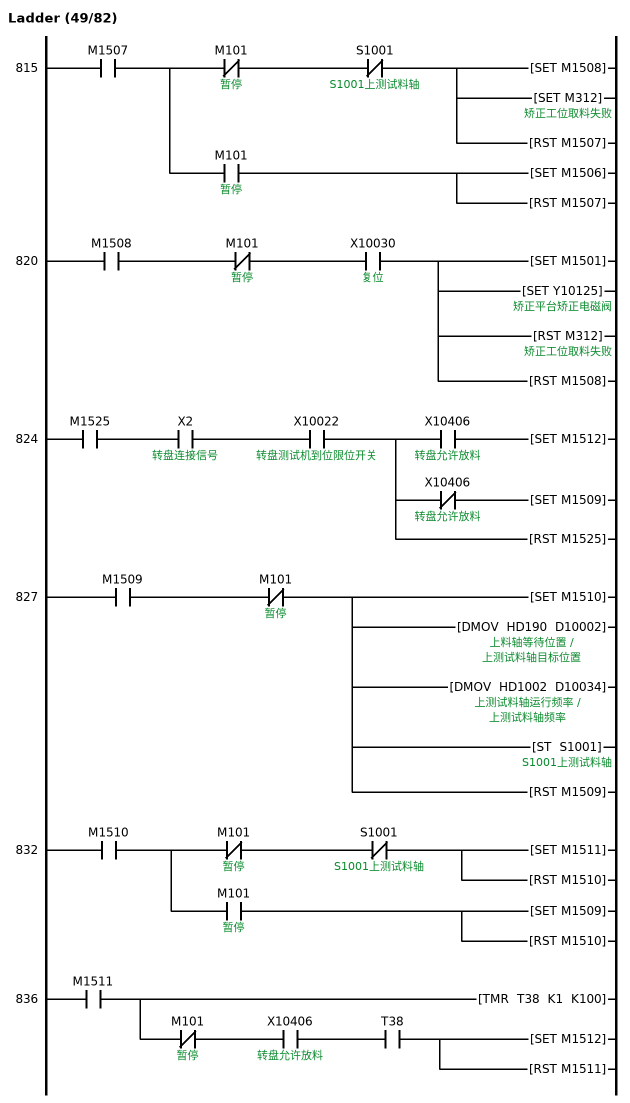
[picture p48: Ladder rows 815-836]
LD     M1507
MPS
ANI    M101	; 暂停
ANI    S1001	; S1001上测试料轴
SET    M1508
SET    M312	; 矫正工位取料失败
RST    M1507
MPP
AND    M101	; 暂停
SET    M1506
RST    M1507
LD     M1508
ANI    M101	; 暂停
AND    X10030	; 复位
SET    M1501
SET    Y10125	; 矫正平台矫正电磁阀
RST    M312	; 矫正工位取料失败
RST    M1508
LD     M1525
AND    X2	; 转盘连接信号
AND    X10022	; 转盘测试机到位限位开关
MPS
AND    X10406	; 转盘允许放料
SET    M1512
MRD
ANI    X10406	; 转盘允许放料
SET    M1509
MPP
RST    M1525
LD     M1509
ANI    M101	; 暂停
SET    M1510
DMOV   HD190 D10002	; 上料轴等待位置 / 上测试料轴目标位置
DMOV   HD1002 D10034	; 上测试料轴运行频率 / 上测试料轴频率
ST     S1001	; S1001上测试料轴
RST    M1509
LD     M1510
MPS
ANI    M101	; 暂停
ANI    S1001	; S1001上测试料轴
SET    M1511
RST    M1510
MPP
AND    M101	; 暂停
SET    M1509
RST    M1510
LD     M1511
TMR    T38 K1 K100
ANI    M101	; 暂停
AND    X10406	; 转盘允许放料
AND    T38
SET    M1512
RST    M1511

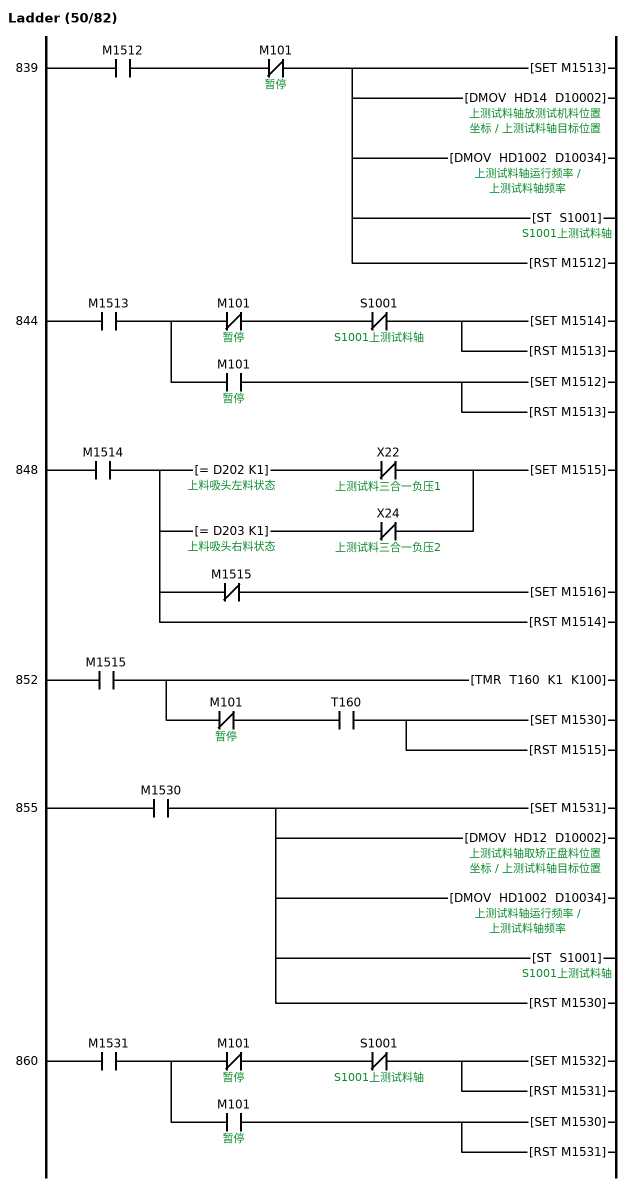
LD     M1512
ANI    M101	; 暂停
SET    M1513
DMOV   HD14 D10002	; 上测试料轴放测试机料位置坐标 / 上测试料轴目标位置
DMOV   HD1002 D10034	; 上测试料轴运行频率 / 上测试料轴频率
ST     S1001	; S1001上测试料轴
RST    M1512
LD     M1513
MPS
ANI    M101	; 暂停
ANI    S1001	; S1001上测试料轴
SET    M1514
RST    M1513
MPP
AND    M101	; 暂停
SET    M1512
RST    M1513
LD     M1514
MPS
LD=    D202 K1	; 上料吸头左料状态
ANI    X22	; 上测试料三合一负压1
LD=    D203 K1	; 上料吸头右料状态
ANI    X24	; 上测试料三合一负压2
ORB
ANB
SET    M1515
MRD
ANI    M1515
SET    M1516
MPP
RST    M1514
LD     M1515
TMR    T160 K1 K100
ANI    M101	; 暂停
AND    T160
SET    M1530
RST    M1515
LD     M1530
SET    M1531
DMOV   HD12 D10002	; 上测试料轴取矫正盘料位置坐标 / 上测试料轴目标位置
DMOV   HD1002 D10034	; 上测试料轴运行频率 / 上测试料轴频率
ST     S1001	; S1001上测试料轴
RST    M1530
LD     M1531
MPS
ANI    M101	; 暂停
ANI    S1001	; S1001上测试料轴
SET    M1532
RST    M1531
MPP
AND    M101	; 暂停
SET    M1530
RST    M1531

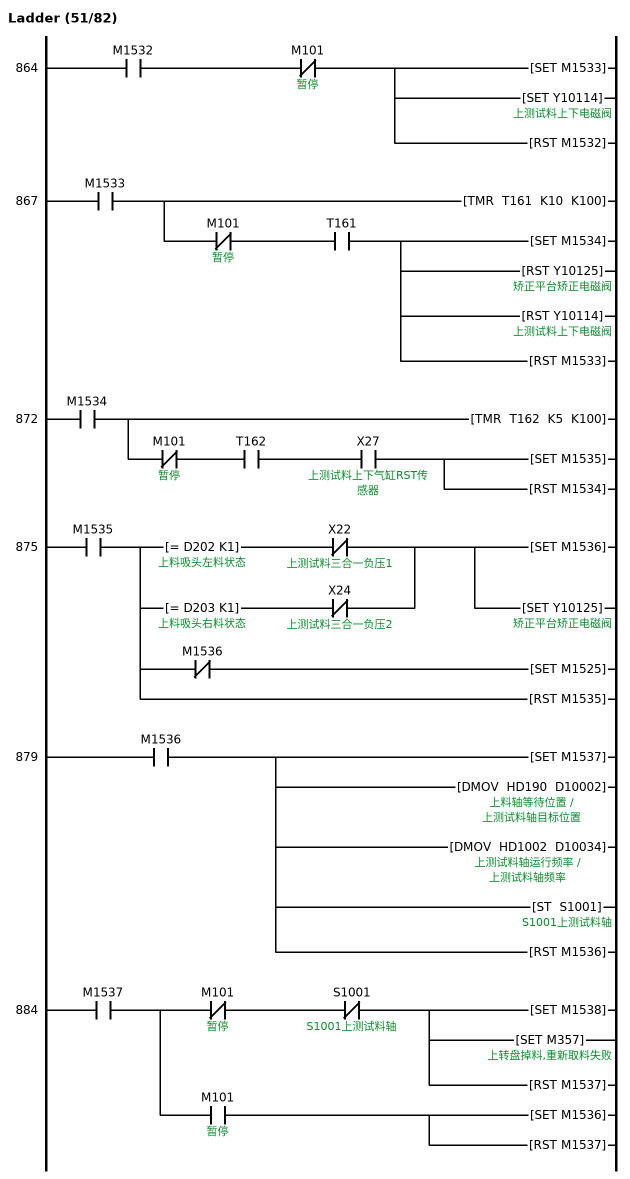
LD     M1532
ANI    M101	; 暂停
SET    M1533
SET    Y10114	; 上测试料上下电磁阀
RST    M1532
LD     M1533
TMR    T161 K10 K100
ANI    M101	; 暂停
AND    T161
SET    M1534
RST    Y10125	; 矫正平台矫正电磁阀
RST    Y10114	; 上测试料上下电磁阀
RST    M1533
LD     M1534
TMR    T162 K5 K100
ANI    M101	; 暂停
AND    T162
AND    X27	; 上测试料上下气缸RST传感器
SET    M1535
RST    M1534
LD     M1535
MPS
LD=    D202 K1	; 上料吸头左料状态
ANI    X22	; 上测试料三合一负压1
LD=    D203 K1	; 上料吸头右料状态
ANI    X24	; 上测试料三合一负压2
ORB
ANB
SET    M1536
SET    Y10125	; 矫正平台矫正电磁阀
MRD
ANI    M1536
SET    M1525
MPP
RST    M1535
LD     M1536
SET    M1537
DMOV   HD190 D10002	; 上料轴等待位置 / 上测试料轴目标位置
DMOV   HD1002 D10034	; 上测试料轴运行频率 / 上测试料轴频率
ST     S1001	; S1001上测试料轴
RST    M1536
LD     M1537
MPS
ANI    M101	; 暂停
ANI    S1001	; S1001上测试料轴
SET    M1538
SET    M357	; 上转盘掉料,重新取料失败
RST    M1537
MPP
AND    M101	; 暂停
SET    M1536
RST    M1537

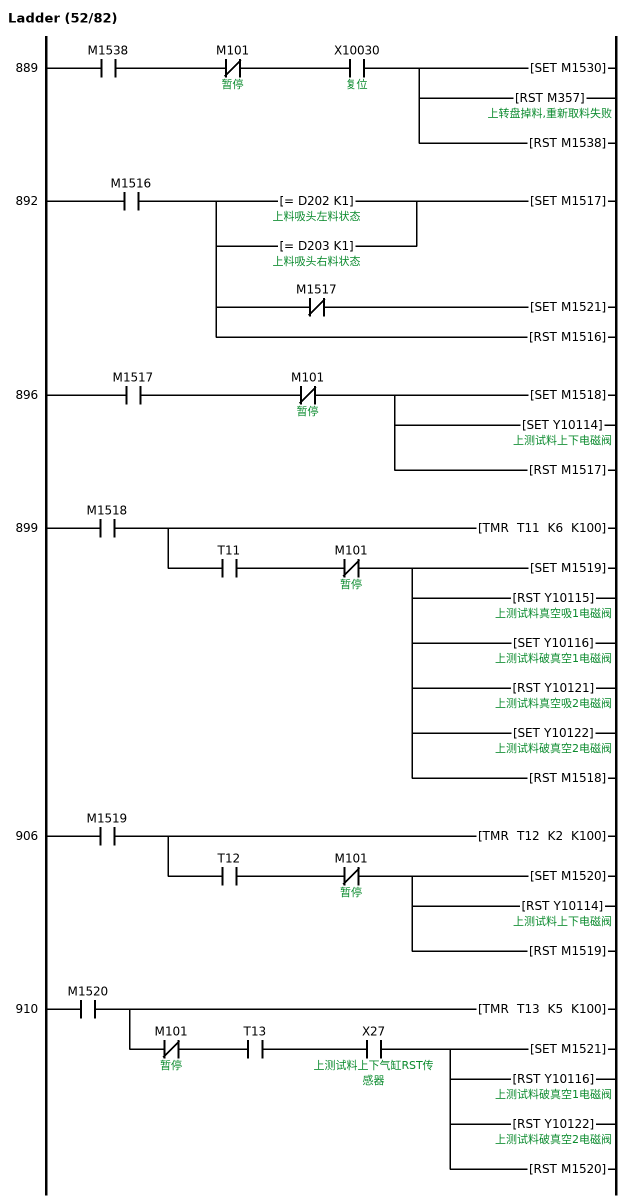
LD     M1538
ANI    M101	; 暂停
AND    X10030	; 复位
SET    M1530
RST    M357	; 上转盘掉料,重新取料失败
RST    M1538
LD     M1516
MPS
LD=    D202 K1	; 上料吸头左料状态
OR=    D203 K1	; 上料吸头右料状态
ANB
SET    M1517
MRD
ANI    M1517
SET    M1521
MPP
RST    M1516
LD     M1517
ANI    M101	; 暂停
SET    M1518
SET    Y10114	; 上测试料上下电磁阀
RST    M1517
LD     M1518
TMR    T11 K6 K100
AND    T11
ANI    M101	; 暂停
SET    M1519
RST    Y10115	; 上测试料真空吸1电磁阀
SET    Y10116	; 上测试料破真空1电磁阀
RST    Y10121	; 上测试料真空吸2电磁阀
SET    Y10122	; 上测试料破真空2电磁阀
RST    M1518
LD     M1519
TMR    T12 K2 K100
AND    T12
ANI    M101	; 暂停
SET    M1520
RST    Y10114	; 上测试料上下电磁阀
RST    M1519
LD     M1520
TMR    T13 K5 K100
ANI    M101	; 暂停
AND    T13
AND    X27	; 上测试料上下气缸RST传感器
SET    M1521
RST    Y10116	; 上测试料破真空1电磁阀
RST    Y10122	; 上测试料破真空2电磁阀
RST    M1520

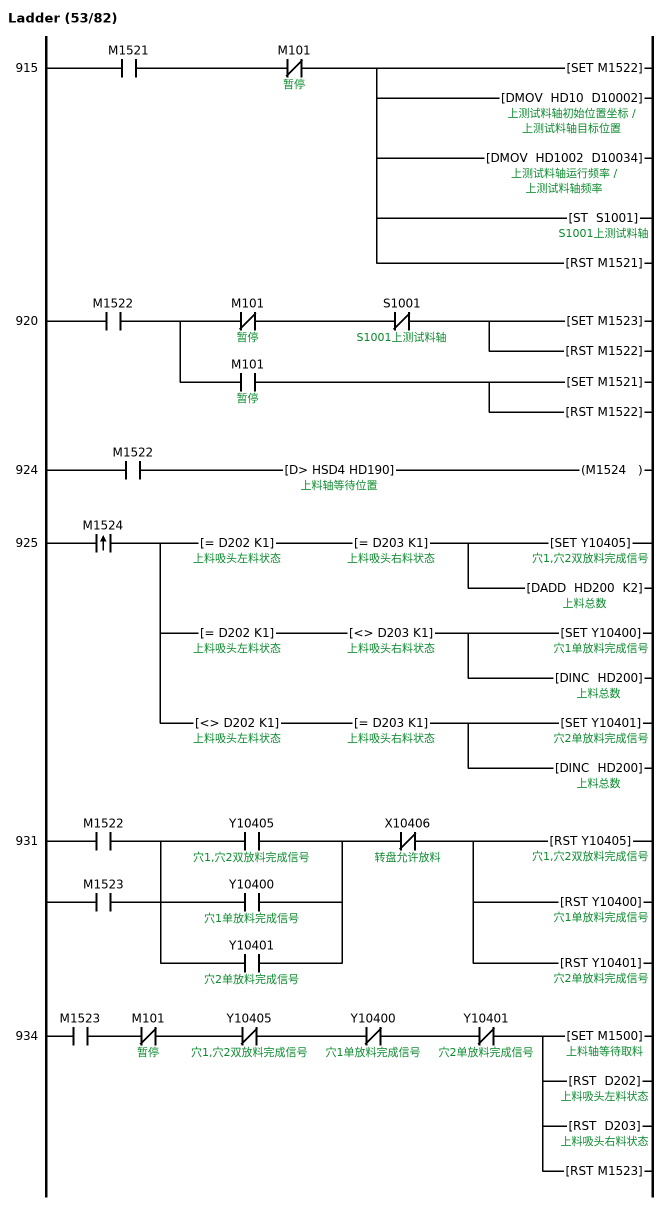
LD     M1521
ANI    M101	; 暂停
SET    M1522
DMOV   HD10 D10002	; 上测试料轴初始位置坐标 / 上测试料轴目标位置
DMOV   HD1002 D10034	; 上测试料轴运行频率 / 上测试料轴频率
ST     S1001	; S1001上测试料轴
RST    M1521
LD     M1522
MPS
ANI    M101	; 暂停
ANI    S1001	; S1001上测试料轴
SET    M1523
RST    M1522
MPP
AND    M101	; 暂停
SET    M1521
RST    M1522
LD     M1522
DAND>  HSD4 HD190	; 上料轴等待位置
OUT    M1524
LDP    M1524
MPS
AND=   D202 K1	; 上料吸头左料状态
AND=   D203 K1	; 上料吸头右料状态
SET    Y10405	; 穴1,穴2双放料完成信号
DADD   HD200 K2	; 上料总数
MRD
AND=   D202 K1	; 上料吸头左料状态
AND<>  D203 K1	; 上料吸头右料状态
SET    Y10400	; 穴1单放料完成信号
DINC   HD200	; 上料总数
MPP
AND<>  D202 K1	; 上料吸头左料状态
AND=   D203 K1	; 上料吸头右料状态
SET    Y10401	; 穴2单放料完成信号
DINC   HD200	; 上料总数
LD     M1522
OR     M1523
LD     Y10405	; 穴1,穴2双放料完成信号
OR     Y10400	; 穴1单放料完成信号
OR     Y10401	; 穴2单放料完成信号
ANB
ANI    X10406	; 转盘允许放料
RST    Y10405	; 穴1,穴2双放料完成信号
RST    Y10400	; 穴1单放料完成信号
RST    Y10401	; 穴2单放料完成信号
LD     M1523
ANI    M101	; 暂停
ANI    Y10405	; 穴1,穴2双放料完成信号
ANI    Y10400	; 穴1单放料完成信号
ANI    Y10401	; 穴2单放料完成信号
SET    M1500	; 上料轴等待取料
RST    D202	; 上料吸头左料状态
RST    D203	; 上料吸头右料状态
RST    M1523

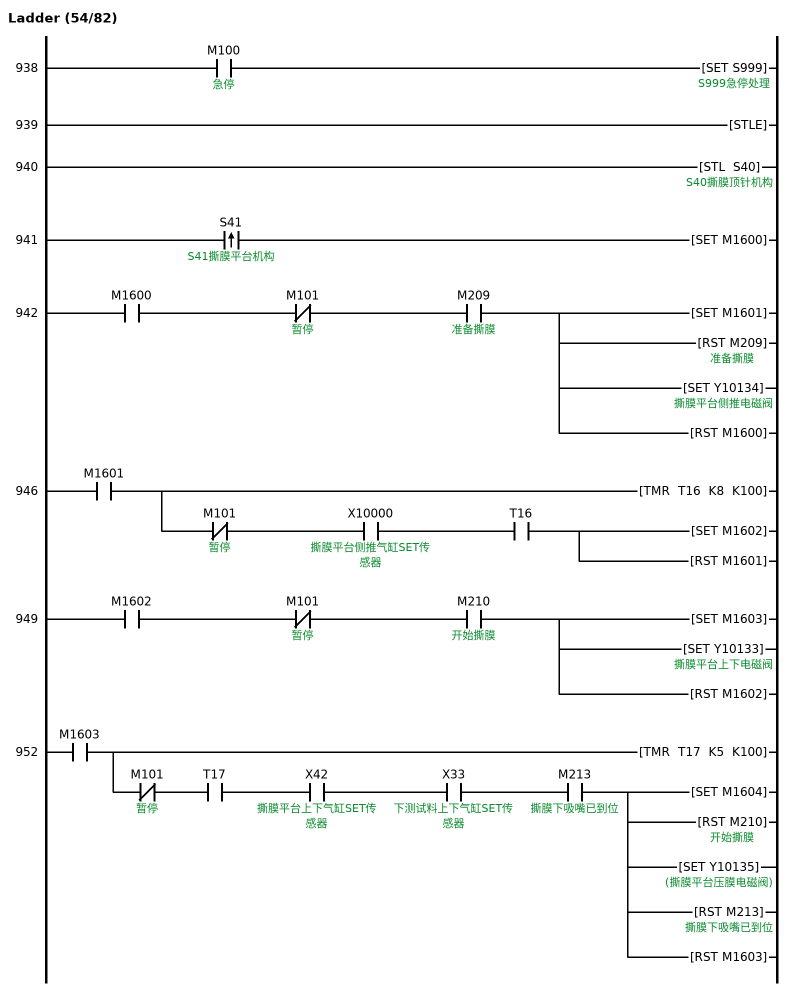
LD     M100	; 急停
SET    S999	; S999急停处理
STLE
STL    S40	; S40撕膜顶针机构
LDP    S41	; S41撕膜平台机构
SET    M1600
LD     M1600
ANI    M101	; 暂停
AND    M209	; 准备撕膜
SET    M1601
RST    M209	; 准备撕膜
SET    Y10134	; 撕膜平台侧推电磁阀
RST    M1600
LD     M1601
TMR    T16 K8 K100
ANI    M101	; 暂停
AND    X10000	; 撕膜平台侧推气缸SET传感器
AND    T16
SET    M1602
RST    M1601
LD     M1602
ANI    M101	; 暂停
AND    M210	; 开始撕膜
SET    M1603
SET    Y10133	; 撕膜平台上下电磁阀
RST    M1602
LD     M1603
TMR    T17 K5 K100
ANI    M101	; 暂停
AND    T17
AND    X42	; 撕膜平台上下气缸SET传感器
AND    X33	; 下测试料上下气缸SET传感器
AND    M213	; 撕膜下吸嘴已到位
SET    M1604
RST    M210	; 开始撕膜
SET    Y10135	; (撕膜平台压膜电磁阀)
RST    M213	; 撕膜下吸嘴已到位
RST    M1603

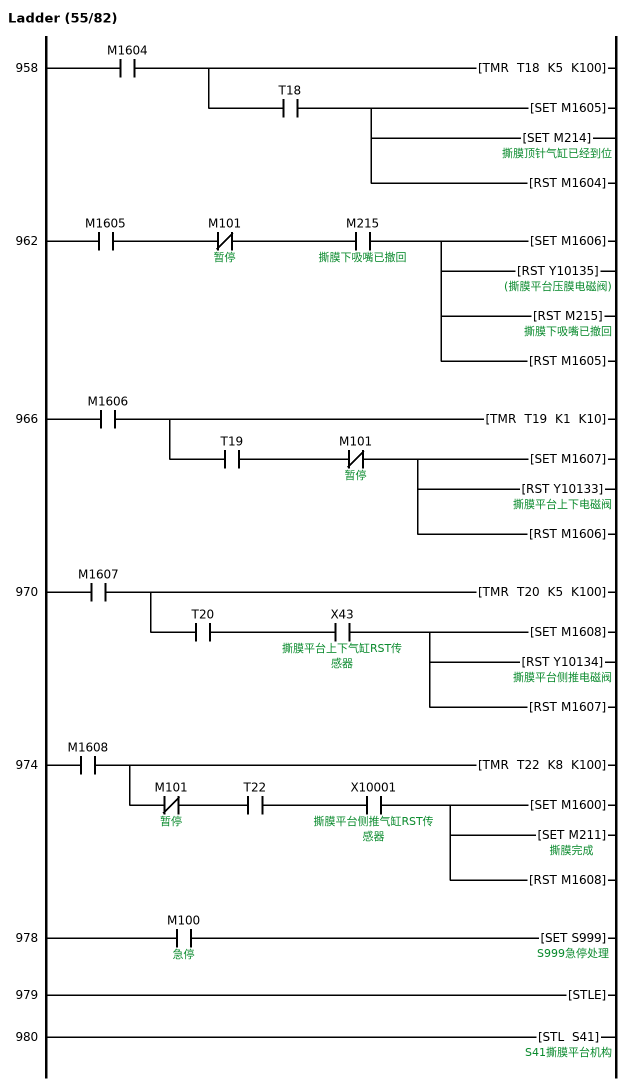
LD     M1604
TMR    T18 K5 K100
AND    T18
SET    M1605
SET    M214	; 撕膜顶针气缸已经到位
RST    M1604
LD     M1605
ANI    M101	; 暂停
AND    M215	; 撕膜下吸嘴已撤回
SET    M1606
RST    Y10135	; (撕膜平台压膜电磁阀)
RST    M215	; 撕膜下吸嘴已撤回
RST    M1605
LD     M1606
TMR    T19 K1 K10
AND    T19
ANI    M101	; 暂停
SET    M1607
RST    Y10133	; 撕膜平台上下电磁阀
RST    M1606
LD     M1607
TMR    T20 K5 K100
AND    T20
AND    X43	; 撕膜平台上下气缸RST传感器
SET    M1608
RST    Y10134	; 撕膜平台侧推电磁阀
RST    M1607
LD     M1608
TMR    T22 K8 K100
ANI    M101	; 暂停
AND    T22
AND    X10001	; 撕膜平台侧推气缸RST传感器
SET    M1600
SET    M211	; 撕膜完成
RST    M1608
LD     M100	; 急停
SET    S999	; S999急停处理
STLE
STL    S41	; S41撕膜平台机构

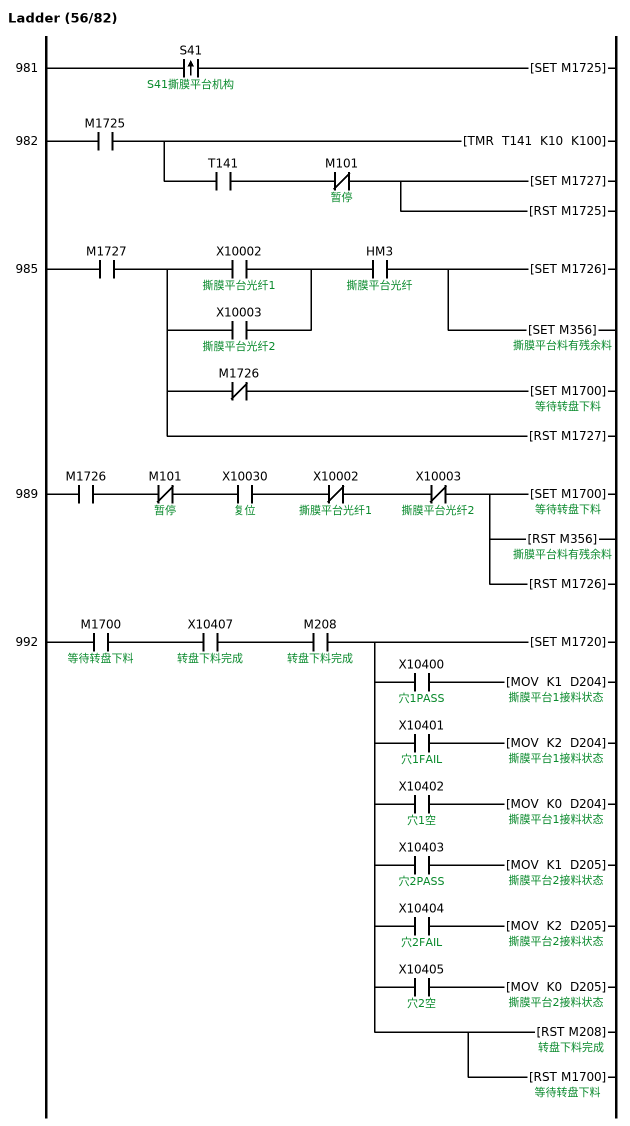
LDP    S41	; S41撕膜平台机构
SET    M1725
LD     M1725
TMR    T141 K10 K100
AND    T141
ANI    M101	; 暂停
SET    M1727
RST    M1725
LD     M1727
MPS
LD     X10002	; 撕膜平台光纤1
OR     X10003	; 撕膜平台光纤2
ANB
AND    HM3	; 撕膜平台光纤
SET    M1726
SET    M356	; 撕膜平台料有残余料
MRD
ANI    M1726
SET    M1700	; 等待转盘下料
MPP
RST    M1727
LD     M1726
ANI    M101	; 暂停
AND    X10030	; 复位
ANI    X10002	; 撕膜平台光纤1
ANI    X10003	; 撕膜平台光纤2
SET    M1700	; 等待转盘下料
RST    M356	; 撕膜平台料有残余料
RST    M1726
LD     M1700	; 等待转盘下料
AND    X10407	; 转盘下料完成
AND    M208	; 转盘下料完成
SET    M1720
MPS
AND    X10400	; 穴1PASS
MOV    K1 D204	; 撕膜平台1接料状态
MRD
AND    X10401	; 穴1FAIL
MOV    K2 D204	; 撕膜平台1接料状态
MRD
AND    X10402	; 穴1空
MOV    K0 D204	; 撕膜平台1接料状态
MRD
AND    X10403	; 穴2PASS
MOV    K1 D205	; 撕膜平台2接料状态
MRD
AND    X10404	; 穴2FAIL
MOV    K2 D205	; 撕膜平台2接料状态
MRD
AND    X10405	; 穴2空
MOV    K0 D205	; 撕膜平台2接料状态
MPP
RST    M208	; 转盘下料完成
RST    M1700	; 等待转盘下料

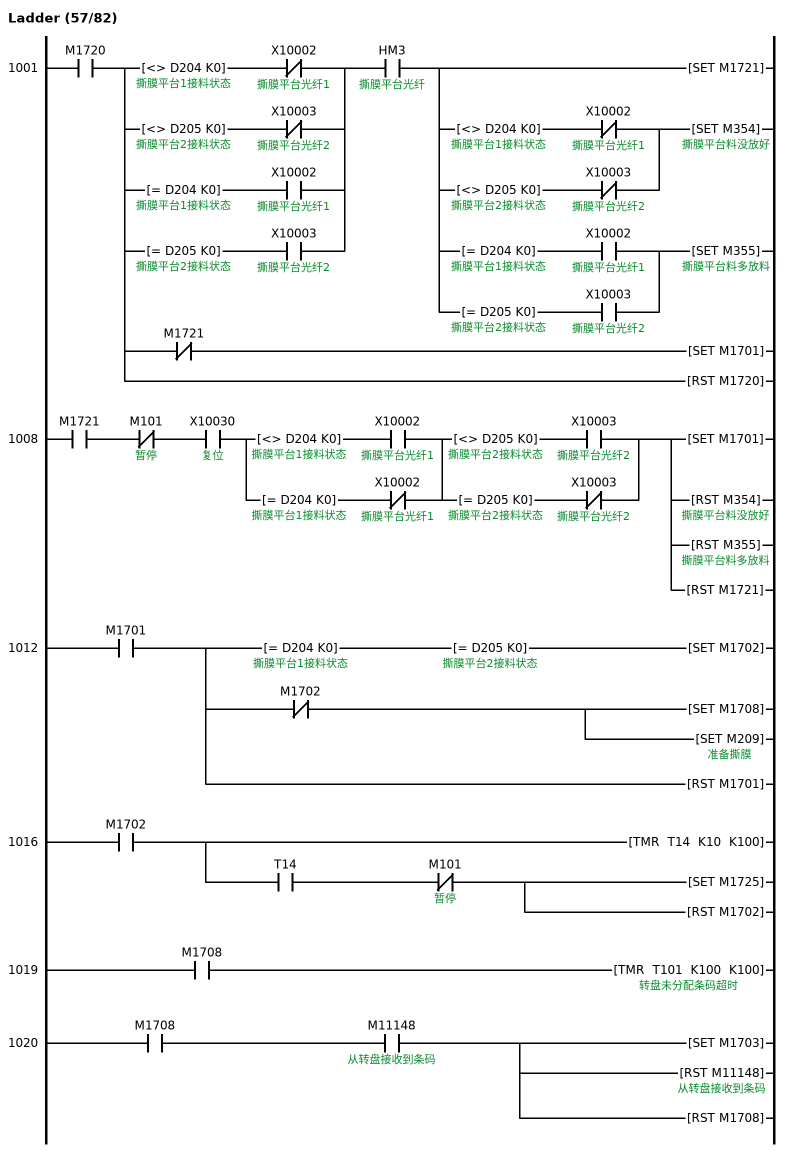
LD     M1720
MPS
LD<>   D204 K0	; 撕膜平台1接料状态
ANI    X10002	; 撕膜平台光纤1
LD<>   D205 K0	; 撕膜平台2接料状态
ANI    X10003	; 撕膜平台光纤2
ORB
LD=    D204 K0	; 撕膜平台1接料状态
AND    X10002	; 撕膜平台光纤1
ORB
LD=    D205 K0	; 撕膜平台2接料状态
AND    X10003	; 撕膜平台光纤2
ORB
ANB
AND    HM3	; 撕膜平台光纤
SET    M1721
MPS
LD<>   D204 K0	; 撕膜平台1接料状态
ANI    X10002	; 撕膜平台光纤1
LD<>   D205 K0	; 撕膜平台2接料状态
ANI    X10003	; 撕膜平台光纤2
ORB
ANB
SET    M354	; 撕膜平台料没放好
MPP
LD=    D204 K0	; 撕膜平台1接料状态
AND    X10002	; 撕膜平台光纤1
LD=    D205 K0	; 撕膜平台2接料状态
AND    X10003	; 撕膜平台光纤2
ORB
ANB
SET    M355	; 撕膜平台料多放料
MRD
ANI    M1721
SET    M1701
MPP
RST    M1720
LD     M1721
ANI    M101	; 暂停
AND    X10030	; 复位
LD<>   D204 K0	; 撕膜平台1接料状态
AND    X10002	; 撕膜平台光纤1
LD=    D204 K0	; 撕膜平台1接料状态
ANI    X10002	; 撕膜平台光纤1
ORB
ANB
LD<>   D205 K0	; 撕膜平台2接料状态
AND    X10003	; 撕膜平台光纤2
LD=    D205 K0	; 撕膜平台2接料状态
ANI    X10003	; 撕膜平台光纤2
ORB
ANB
SET    M1701
RST    M354	; 撕膜平台料没放好
RST    M355	; 撕膜平台料多放料
RST    M1721
LD     M1701
MPS
AND=   D204 K0	; 撕膜平台1接料状态
AND=   D205 K0	; 撕膜平台2接料状态
SET    M1702
MRD
ANI    M1702
SET    M1708
SET    M209	; 准备撕膜
MPP
RST    M1701
LD     M1702
TMR    T14 K10 K100
AND    T14
ANI    M101	; 暂停
SET    M1725
RST    M1702
LD     M1708
TMR    T101 K100 K100	; 转盘未分配条码超时
LD     M1708
AND    M11148	; 从转盘接收到条码
SET    M1703
RST    M11148	; 从转盘接收到条码
RST    M1708

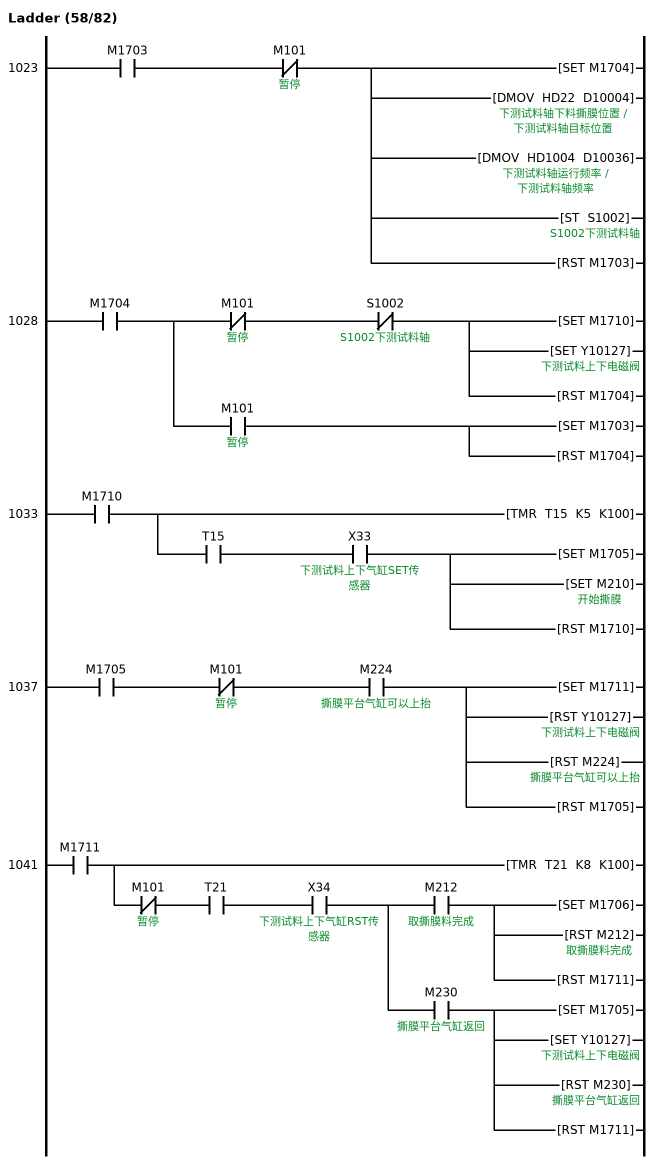
LD     M1703
ANI    M101	; 暂停
SET    M1704
DMOV   HD22 D10004	; 下测试料轴下料撕膜位置 / 下测试料轴目标位置
DMOV   HD1004 D10036	; 下测试料轴运行频率 / 下测试料轴频率
ST     S1002	; S1002下测试料轴
RST    M1703
LD     M1704
MPS
ANI    M101	; 暂停
ANI    S1002	; S1002下测试料轴
SET    M1710
SET    Y10127	; 下测试料上下电磁阀
RST    M1704
MPP
AND    M101	; 暂停
SET    M1703
RST    M1704
LD     M1710
TMR    T15 K5 K100
AND    T15
AND    X33	; 下测试料上下气缸SET传感器
SET    M1705
SET    M210	; 开始撕膜
RST    M1710
LD     M1705
ANI    M101	; 暂停
AND    M224	; 撕膜平台气缸可以上抬
SET    M1711
RST    Y10127	; 下测试料上下电磁阀
RST    M224	; 撕膜平台气缸可以上抬
RST    M1705
LD     M1711
TMR    T21 K8 K100
ANI    M101	; 暂停
AND    T21
AND    X34	; 下测试料上下气缸RST传感器
MPS
AND    M212	; 取撕膜料完成
SET    M1706
RST    M212	; 取撕膜料完成
RST    M1711
MPP
AND    M230	; 撕膜平台气缸返回
SET    M1705
SET    Y10127	; 下测试料上下电磁阀
RST    M230	; 撕膜平台气缸返回
RST    M1711

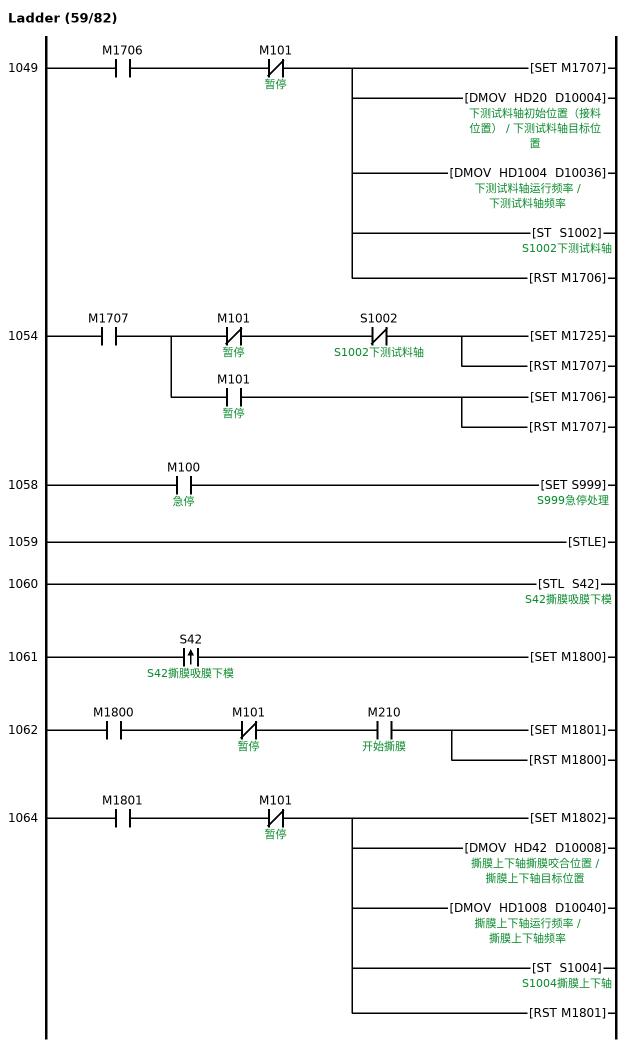
LD     M1706
ANI    M101	; 暂停
SET    M1707
DMOV   HD20 D10004	; 下测试料轴初始位置（接料位置） / 下测试料轴目标位置
DMOV   HD1004 D10036	; 下测试料轴运行频率 / 下测试料轴频率
ST     S1002	; S1002下测试料轴
RST    M1706
LD     M1707
MPS
ANI    M101	; 暂停
ANI    S1002	; S1002下测试料轴
SET    M1725
RST    M1707
MPP
AND    M101	; 暂停
SET    M1706
RST    M1707
LD     M100	; 急停
SET    S999	; S999急停处理
STLE
STL    S42	; S42撕膜吸膜下模
LDP    S42	; S42撕膜吸膜下模
SET    M1800
LD     M1800
ANI    M101	; 暂停
AND    M210	; 开始撕膜
SET    M1801
RST    M1800
LD     M1801
ANI    M101	; 暂停
SET    M1802
DMOV   HD42 D10008	; 撕膜上下轴撕膜咬合位置 / 撕膜上下轴目标位置
DMOV   HD1008 D10040	; 撕膜上下轴运行频率 / 撕膜上下轴频率
ST     S1004	; S1004撕膜上下轴
RST    M1801

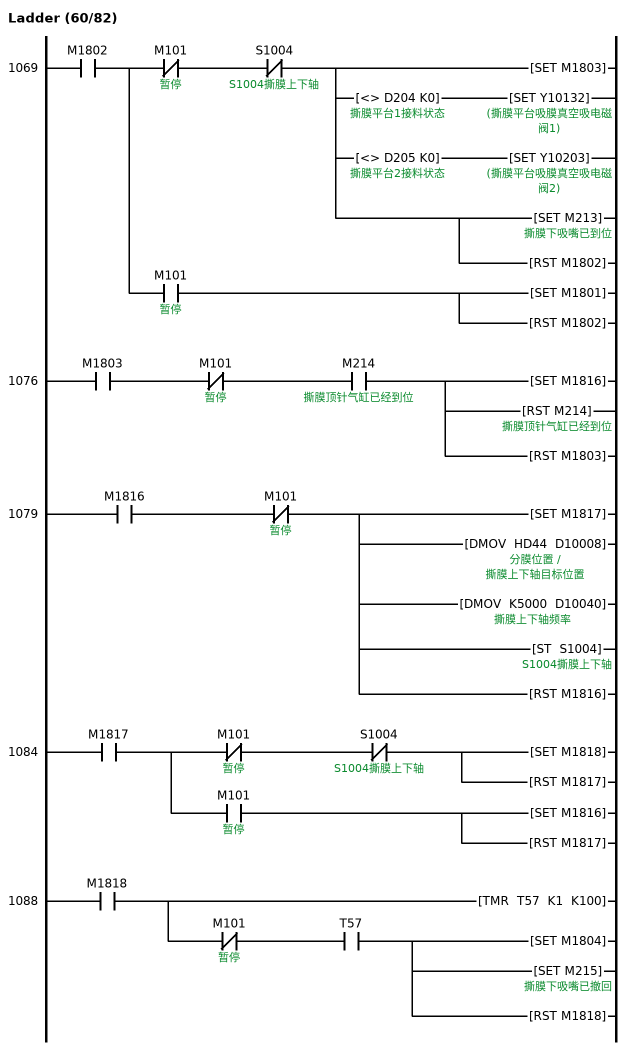
LD     M1802
MPS
ANI    M101	; 暂停
ANI    S1004	; S1004撕膜上下轴
SET    M1803
MPS
AND<>  D204 K0	; 撕膜平台1接料状态
SET    Y10132	; (撕膜平台吸膜真空吸电磁阀1)
MRD
AND<>  D205 K0	; 撕膜平台2接料状态
SET    Y10203	; (撕膜平台吸膜真空吸电磁阀2)
MPP
SET    M213	; 撕膜下吸嘴已到位
RST    M1802
MPP
AND    M101	; 暂停
SET    M1801
RST    M1802
LD     M1803
ANI    M101	; 暂停
AND    M214	; 撕膜顶针气缸已经到位
SET    M1816
RST    M214	; 撕膜顶针气缸已经到位
RST    M1803
LD     M1816
ANI    M101	; 暂停
SET    M1817
DMOV   HD44 D10008	; 分膜位置 / 撕膜上下轴目标位置
DMOV   K5000 D10040	; 撕膜上下轴频率
ST     S1004	; S1004撕膜上下轴
RST    M1816
LD     M1817
MPS
ANI    M101	; 暂停
ANI    S1004	; S1004撕膜上下轴
SET    M1818
RST    M1817
MPP
AND    M101	; 暂停
SET    M1816
RST    M1817
LD     M1818
TMR    T57 K1 K100
ANI    M101	; 暂停
AND    T57
SET    M1804
SET    M215	; 撕膜下吸嘴已撤回
RST    M1818

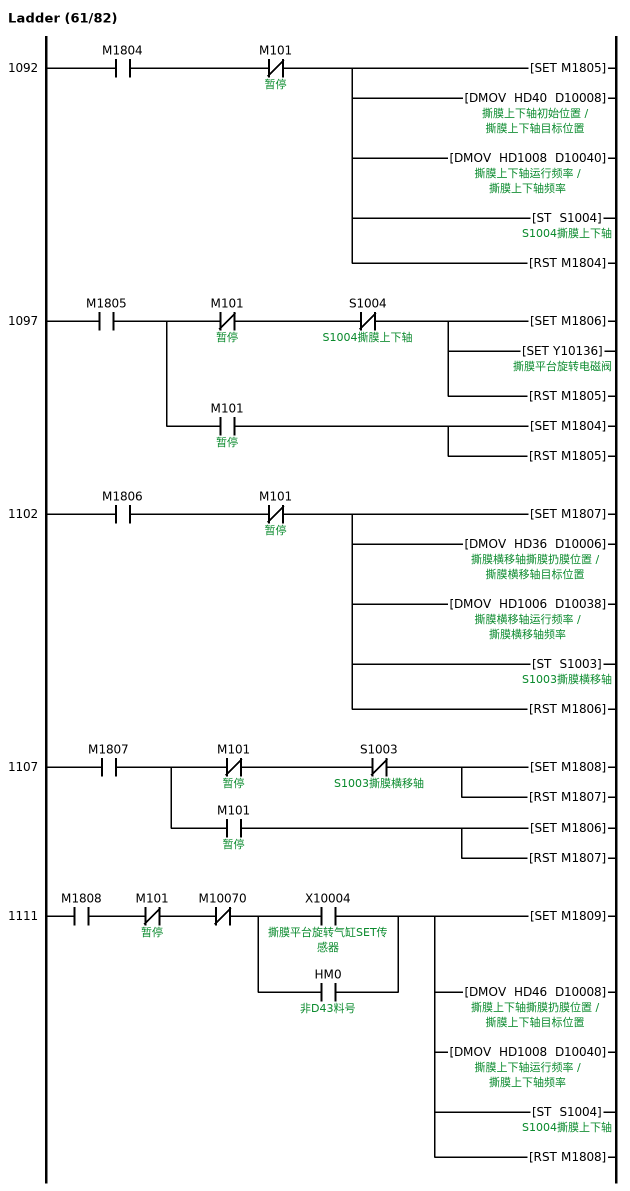
LD     M1804
ANI    M101	; 暂停
SET    M1805
DMOV   HD40 D10008	; 撕膜上下轴初始位置 / 撕膜上下轴目标位置
DMOV   HD1008 D10040	; 撕膜上下轴运行频率 / 撕膜上下轴频率
ST     S1004	; S1004撕膜上下轴
RST    M1804
LD     M1805
MPS
ANI    M101	; 暂停
ANI    S1004	; S1004撕膜上下轴
SET    M1806
SET    Y10136	; 撕膜平台旋转电磁阀
RST    M1805
MPP
AND    M101	; 暂停
SET    M1804
RST    M1805
LD     M1806
ANI    M101	; 暂停
SET    M1807
DMOV   HD36 D10006	; 撕膜横移轴撕膜扔膜位置 / 撕膜横移轴目标位置
DMOV   HD1006 D10038	; 撕膜横移轴运行频率 / 撕膜横移轴频率
ST     S1003	; S1003撕膜横移轴
RST    M1806
LD     M1807
MPS
ANI    M101	; 暂停
ANI    S1003	; S1003撕膜横移轴
SET    M1808
RST    M1807
MPP
AND    M101	; 暂停
SET    M1806
RST    M1807
LD     M1808
ANI    M101	; 暂停
ANI    M10070
LD     X10004	; 撕膜平台旋转气缸SET传感器
OR     HM0	; 非D43料号
ANB
SET    M1809
DMOV   HD46 D10008	; 撕膜上下轴撕膜扔膜位置 / 撕膜上下轴目标位置
DMOV   HD1008 D10040	; 撕膜上下轴运行频率 / 撕膜上下轴频率
ST     S1004	; S1004撕膜上下轴
RST    M1808

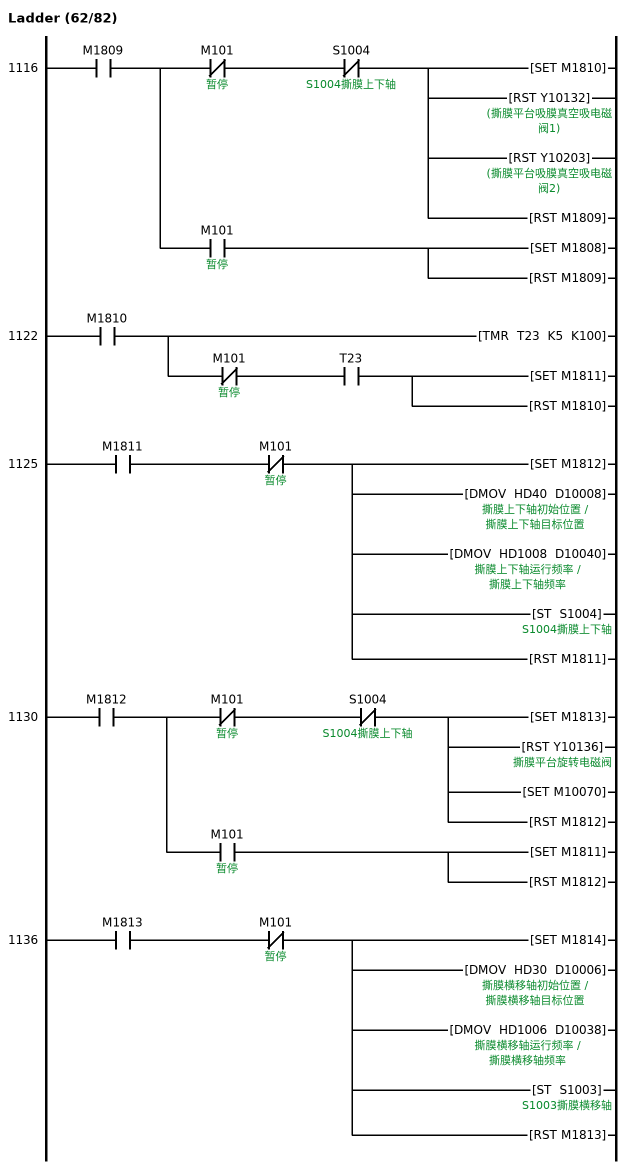
LD     M1809
MPS
ANI    M101	; 暂停
ANI    S1004	; S1004撕膜上下轴
SET    M1810
RST    Y10132	; (撕膜平台吸膜真空吸电磁阀1)
RST    Y10203	; (撕膜平台吸膜真空吸电磁阀2)
RST    M1809
MPP
AND    M101	; 暂停
SET    M1808
RST    M1809
LD     M1810
TMR    T23 K5 K100
ANI    M101	; 暂停
AND    T23
SET    M1811
RST    M1810
LD     M1811
ANI    M101	; 暂停
SET    M1812
DMOV   HD40 D10008	; 撕膜上下轴初始位置 / 撕膜上下轴目标位置
DMOV   HD1008 D10040	; 撕膜上下轴运行频率 / 撕膜上下轴频率
ST     S1004	; S1004撕膜上下轴
RST    M1811
LD     M1812
MPS
ANI    M101	; 暂停
ANI    S1004	; S1004撕膜上下轴
SET    M1813
RST    Y10136	; 撕膜平台旋转电磁阀
SET    M10070
RST    M1812
MPP
AND    M101	; 暂停
SET    M1811
RST    M1812
LD     M1813
ANI    M101	; 暂停
SET    M1814
DMOV   HD30 D10006	; 撕膜横移轴初始位置 / 撕膜横移轴目标位置
DMOV   HD1006 D10038	; 撕膜横移轴运行频率 / 撕膜横移轴频率
ST     S1003	; S1003撕膜横移轴
RST    M1813

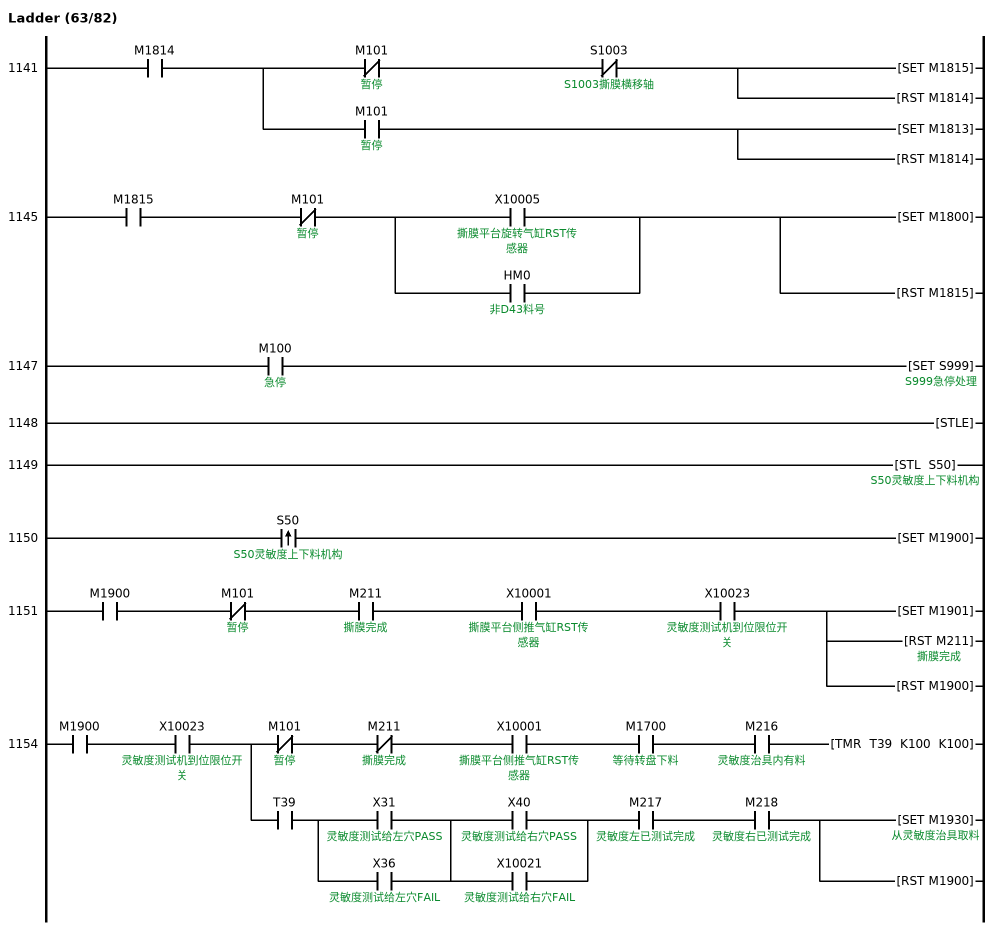
LD     M1814
MPS
ANI    M101	; 暂停
ANI    S1003	; S1003撕膜横移轴
SET    M1815
RST    M1814
MPP
AND    M101	; 暂停
SET    M1813
RST    M1814
LD     M1815
ANI    M101	; 暂停
LD     X10005	; 撕膜平台旋转气缸RST传感器
OR     HM0	; 非D43料号
ANB
SET    M1800
RST    M1815
LD     M100	; 急停
SET    S999	; S999急停处理
STLE
STL    S50	; S50灵敏度上下料机构
LDP    S50	; S50灵敏度上下料机构
SET    M1900
LD     M1900
ANI    M101	; 暂停
AND    M211	; 撕膜完成
AND    X10001	; 撕膜平台侧推气缸RST传感器
AND    X10023	; 灵敏度测试机到位限位开关
SET    M1901
RST    M211	; 撕膜完成
RST    M1900
LD     M1900
AND    X10023	; 灵敏度测试机到位限位开关
MPS
ANI    M101	; 暂停
ANI    M211	; 撕膜完成
AND    X10001	; 撕膜平台侧推气缸RST传感器
AND    M1700	; 等待转盘下料
AND    M216	; 灵敏度治具内有料
TMR    T39 K100 K100
MPP
AND    T39
LD     X31	; 灵敏度测试给左穴PASS
OR     X36	; 灵敏度测试给左穴FAIL
ANB
LD     X40	; 灵敏度测试给右穴PASS
OR     X10021	; 灵敏度测试给右穴FAIL
ANB
AND    M217	; 灵敏度左已测试完成
AND    M218	; 灵敏度右已测试完成
SET    M1930	; 从灵敏度治具取料
RST    M1900

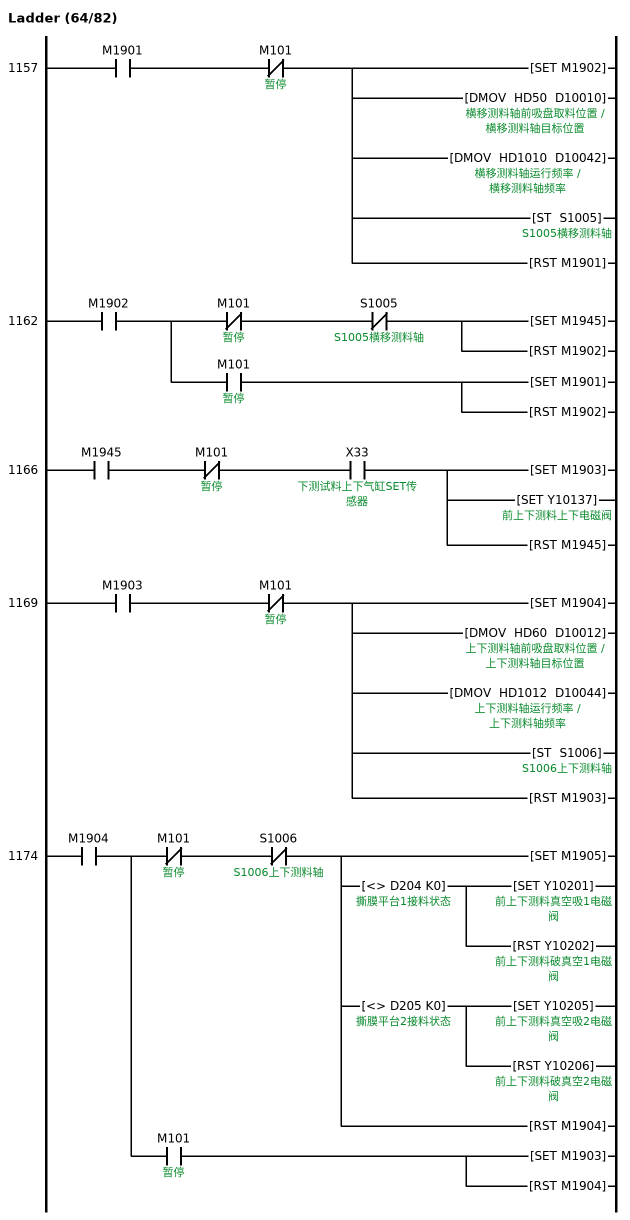
LD     M1901
ANI    M101	; 暂停
SET    M1902
DMOV   HD50 D10010	; 横移测料轴前吸盘取料位置 / 横移测料轴目标位置
DMOV   HD1010 D10042	; 横移测料轴运行频率 / 横移测料轴频率
ST     S1005	; S1005横移测料轴
RST    M1901
LD     M1902
MPS
ANI    M101	; 暂停
ANI    S1005	; S1005横移测料轴
SET    M1945
RST    M1902
MPP
AND    M101	; 暂停
SET    M1901
RST    M1902
LD     M1945
ANI    M101	; 暂停
AND    X33	; 下测试料上下气缸SET传感器
SET    M1903
SET    Y10137	; 前上下测料上下电磁阀
RST    M1945
LD     M1903
ANI    M101	; 暂停
SET    M1904
DMOV   HD60 D10012	; 上下测料轴前吸盘取料位置 / 上下测料轴目标位置
DMOV   HD1012 D10044	; 上下测料轴运行频率 / 上下测料轴频率
ST     S1006	; S1006上下测料轴
RST    M1903
LD     M1904
MPS
ANI    M101	; 暂停
ANI    S1006	; S1006上下测料轴
SET    M1905
MPS
AND<>  D204 K0	; 撕膜平台1接料状态
SET    Y10201	; 前上下测料真空吸1电磁阀
RST    Y10202	; 前上下测料破真空1电磁阀
MRD
AND<>  D205 K0	; 撕膜平台2接料状态
SET    Y10205	; 前上下测料真空吸2电磁阀
RST    Y10206	; 前上下测料破真空2电磁阀
MPP
RST    M1904
MPP
AND    M101	; 暂停
SET    M1903
RST    M1904

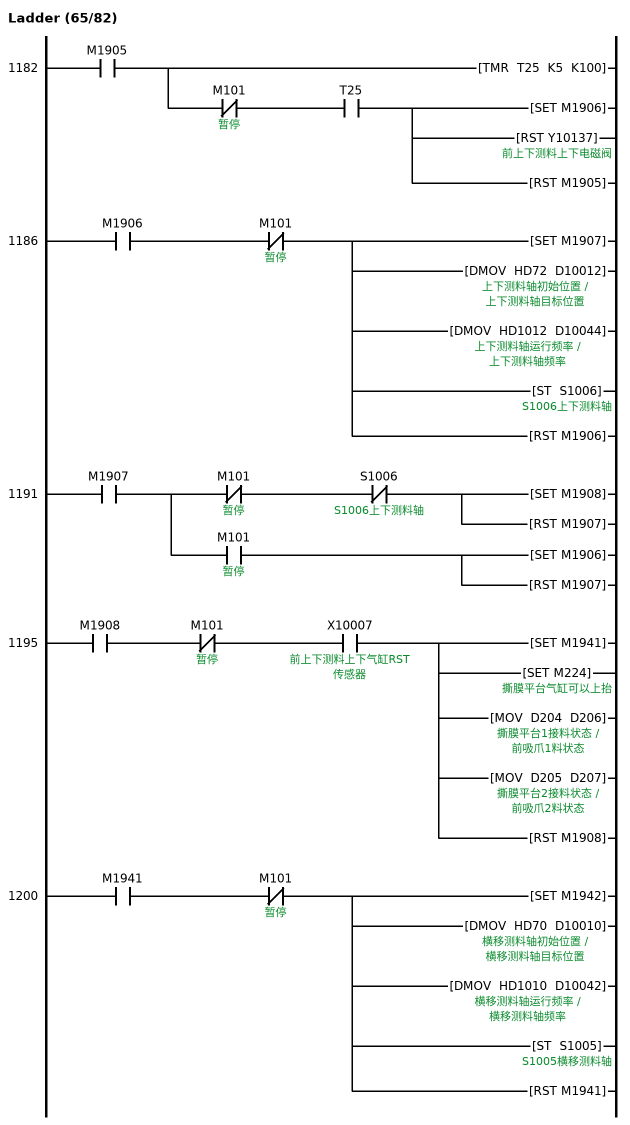
LD     M1905
TMR    T25 K5 K100
ANI    M101	; 暂停
AND    T25
SET    M1906
RST    Y10137	; 前上下测料上下电磁阀
RST    M1905
LD     M1906
ANI    M101	; 暂停
SET    M1907
DMOV   HD72 D10012	; 上下测料轴初始位置 / 上下测料轴目标位置
DMOV   HD1012 D10044	; 上下测料轴运行频率 / 上下测料轴频率
ST     S1006	; S1006上下测料轴
RST    M1906
LD     M1907
MPS
ANI    M101	; 暂停
ANI    S1006	; S1006上下测料轴
SET    M1908
RST    M1907
MPP
AND    M101	; 暂停
SET    M1906
RST    M1907
LD     M1908
ANI    M101	; 暂停
AND    X10007	; 前上下测料上下气缸RST传感器
SET    M1941
SET    M224	; 撕膜平台气缸可以上抬
MOV    D204 D206	; 撕膜平台1接料状态 / 前吸爪1料状态
MOV    D205 D207	; 撕膜平台2接料状态 / 前吸爪2料状态
RST    M1908
LD     M1941
ANI    M101	; 暂停
SET    M1942
DMOV   HD70 D10010	; 横移测料轴初始位置 / 横移测料轴目标位置
DMOV   HD1010 D10042	; 横移测料轴运行频率 / 横移测料轴频率
ST     S1005	; S1005横移测料轴
RST    M1941

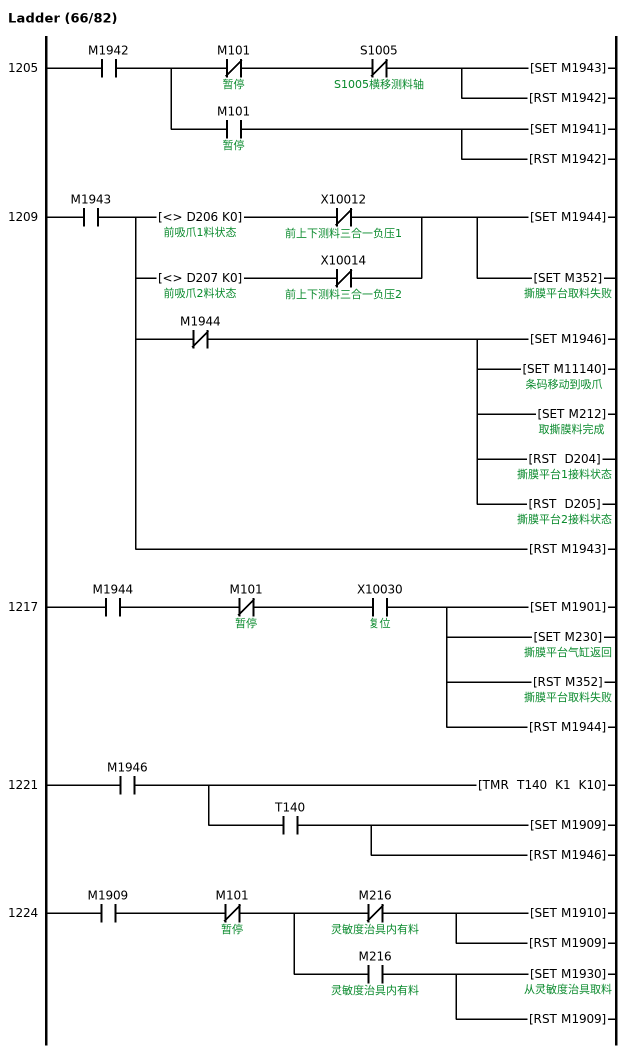
LD     M1942
MPS
ANI    M101	; 暂停
ANI    S1005	; S1005横移测料轴
SET    M1943
RST    M1942
MPP
AND    M101	; 暂停
SET    M1941
RST    M1942
LD     M1943
MPS
LD<>   D206 K0	; 前吸爪1料状态
ANI    X10012	; 前上下测料三合一负压1
LD<>   D207 K0	; 前吸爪2料状态
ANI    X10014	; 前上下测料三合一负压2
ORB
ANB
SET    M1944
SET    M352	; 撕膜平台取料失败
MRD
ANI    M1944
SET    M1946
SET    M11140	; 条码移动到吸爪
SET    M212	; 取撕膜料完成
RST    D204	; 撕膜平台1接料状态
RST    D205	; 撕膜平台2接料状态
MPP
RST    M1943
LD     M1944
ANI    M101	; 暂停
AND    X10030	; 复位
SET    M1901
SET    M230	; 撕膜平台气缸返回
RST    M352	; 撕膜平台取料失败
RST    M1944
LD     M1946
TMR    T140 K1 K10
AND    T140
SET    M1909
RST    M1946
LD     M1909
ANI    M101	; 暂停
MPS
ANI    M216	; 灵敏度治具内有料
SET    M1910
RST    M1909
MPP
AND    M216	; 灵敏度治具内有料
SET    M1930	; 从灵敏度治具取料
RST    M1909

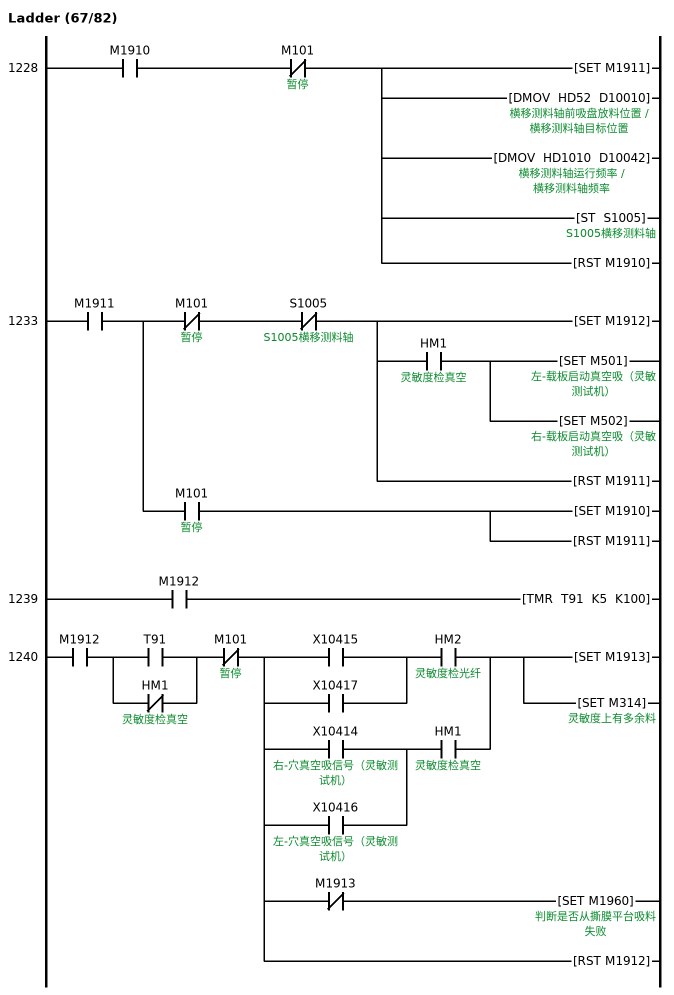
LD     M1910
ANI    M101	; 暂停
SET    M1911
DMOV   HD52 D10010	; 横移测料轴前吸盘放料位置 / 横移测料轴目标位置
DMOV   HD1010 D10042	; 横移测料轴运行频率 / 横移测料轴频率
ST     S1005	; S1005横移测料轴
RST    M1910
LD     M1911
MPS
ANI    M101	; 暂停
ANI    S1005	; S1005横移测料轴
SET    M1912
MPS
AND    HM1	; 灵敏度检真空
SET    M501	; 左-载板启动真空吸（灵敏测试机）
SET    M502	; 右-载板启动真空吸（灵敏测试机）
MPP
RST    M1911
MPP
AND    M101	; 暂停
SET    M1910
RST    M1911
LD     M1912
TMR    T91 K5 K100
LD     M1912
LD     T91
ORI    HM1	; 灵敏度检真空
ANB
ANI    M101	; 暂停
MPS
LD     X10415
OR     X10417
AND    HM2	; 灵敏度检光纤
LD     X10414	; 右-穴真空吸信号（灵敏测试机）
OR     X10416	; 左-穴真空吸信号（灵敏测试机）
AND    HM1	; 灵敏度检真空
ORB
ANB
SET    M1913
SET    M314	; 灵敏度上有多余料
MRD
ANI    M1913
SET    M1960	; 判断是否从撕膜平台吸料失败
MPP
RST    M1912

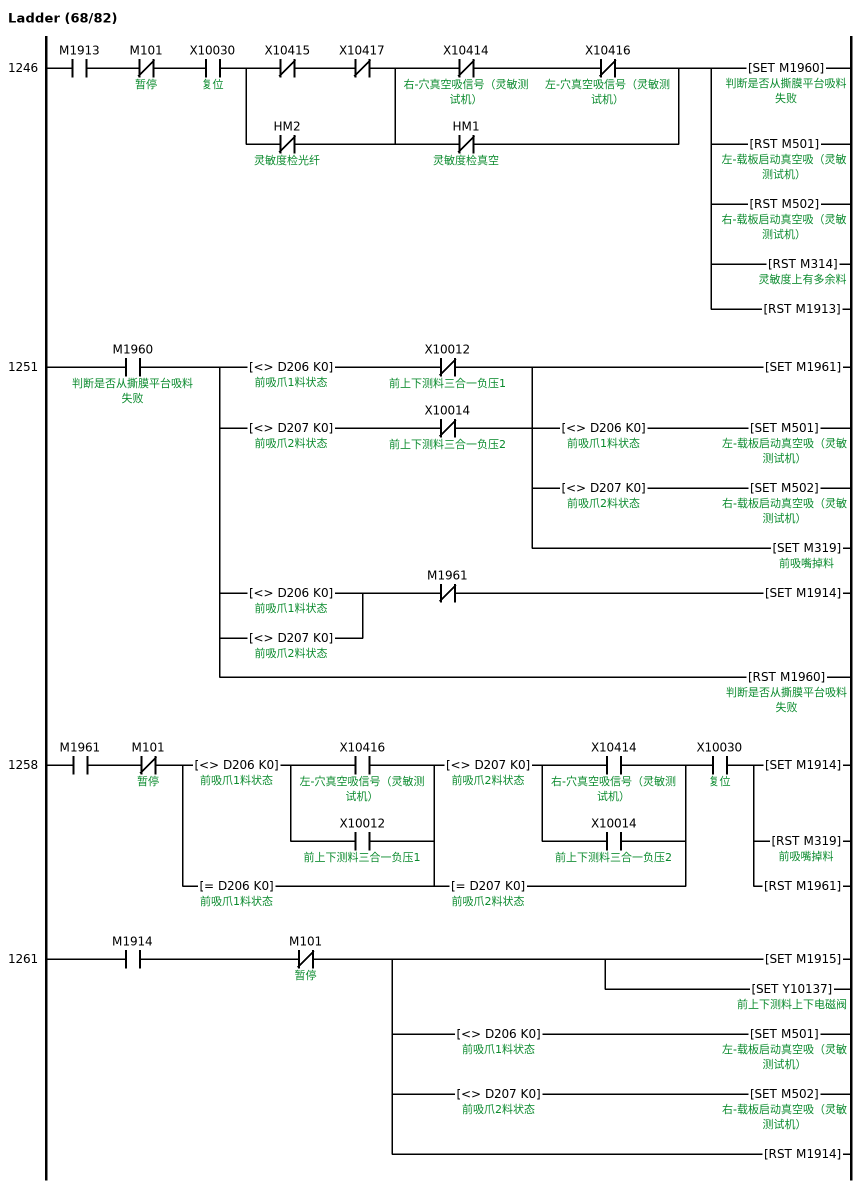
LD     M1913
ANI    M101	; 暂停
AND    X10030	; 复位
LDI    X10415
ANI    X10417
ORI    HM2	; 灵敏度检光纤
ANB
LDI    X10414	; 右-穴真空吸信号（灵敏测试机）
ANI    X10416	; 左-穴真空吸信号（灵敏测试机）
ORI    HM1	; 灵敏度检真空
ANB
SET    M1960	; 判断是否从撕膜平台吸料失败
RST    M501	; 左-载板启动真空吸（灵敏测试机）
RST    M502	; 右-载板启动真空吸（灵敏测试机）
RST    M314	; 灵敏度上有多余料
RST    M1913
LD     M1960	; 判断是否从撕膜平台吸料失败
MPS
LD<>   D206 K0	; 前吸爪1料状态
ANI    X10012	; 前上下测料三合一负压1
LD<>   D207 K0	; 前吸爪2料状态
ANI    X10014	; 前上下测料三合一负压2
ORB
ANB
SET    M1961
MPS
AND<>  D206 K0	; 前吸爪1料状态
SET    M501	; 左-载板启动真空吸（灵敏测试机）
MRD
AND<>  D207 K0	; 前吸爪2料状态
SET    M502	; 右-载板启动真空吸（灵敏测试机）
MPP
SET    M319	; 前吸嘴掉料
MRD
LD<>   D206 K0	; 前吸爪1料状态
OR<>   D207 K0	; 前吸爪2料状态
ANB
ANI    M1961
SET    M1914
MPP
RST    M1960	; 判断是否从撕膜平台吸料失败
LD     M1961
ANI    M101	; 暂停
LD<>   D206 K0	; 前吸爪1料状态
LD     X10416	; 左-穴真空吸信号（灵敏测试机）
OR     X10012	; 前上下测料三合一负压1
ANB
OR=    D206 K0	; 前吸爪1料状态
ANB
LD<>   D207 K0	; 前吸爪2料状态
LD     X10414	; 右-穴真空吸信号（灵敏测试机）
OR     X10014	; 前上下测料三合一负压2
ANB
OR=    D207 K0	; 前吸爪2料状态
ANB
AND    X10030	; 复位
SET    M1914
RST    M319	; 前吸嘴掉料
RST    M1961
LD     M1914
ANI    M101	; 暂停
SET    M1915
SET    Y10137	; 前上下测料上下电磁阀
MPS
AND<>  D206 K0	; 前吸爪1料状态
SET    M501	; 左-载板启动真空吸（灵敏测试机）
MRD
AND<>  D207 K0	; 前吸爪2料状态
SET    M502	; 右-载板启动真空吸（灵敏测试机）
MPP
RST    M1914

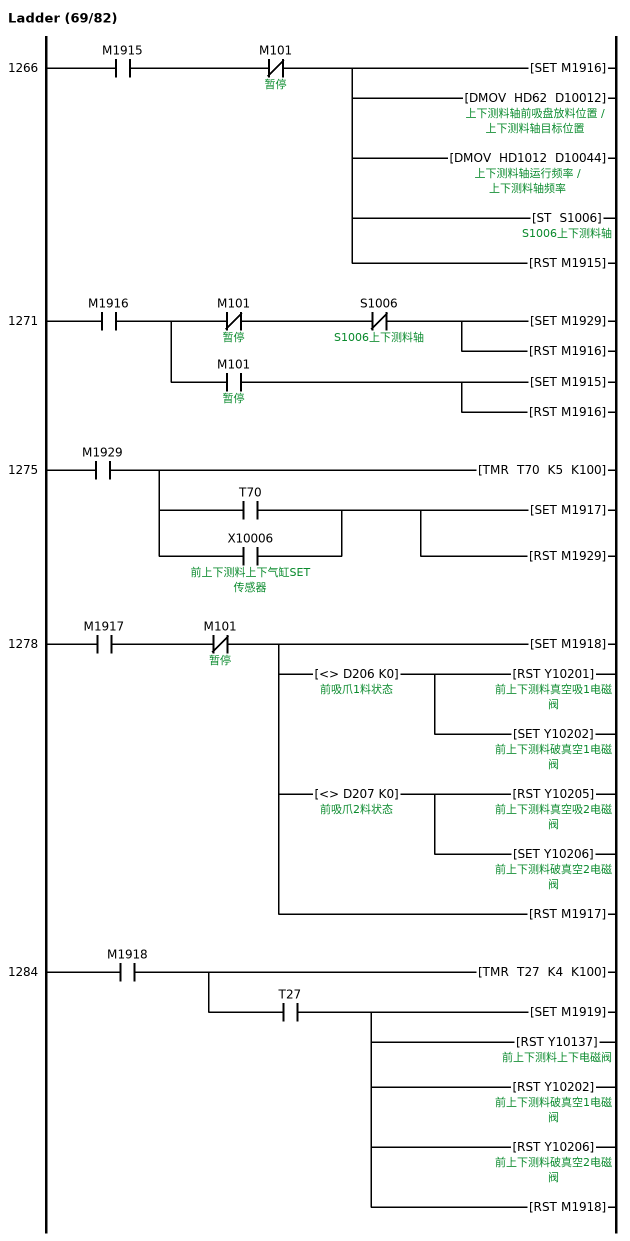
LD     M1915
ANI    M101	; 暂停
SET    M1916
DMOV   HD62 D10012	; 上下测料轴前吸盘放料位置 / 上下测料轴目标位置
DMOV   HD1012 D10044	; 上下测料轴运行频率 / 上下测料轴频率
ST     S1006	; S1006上下测料轴
RST    M1915
LD     M1916
MPS
ANI    M101	; 暂停
ANI    S1006	; S1006上下测料轴
SET    M1929
RST    M1916
MPP
AND    M101	; 暂停
SET    M1915
RST    M1916
LD     M1929
TMR    T70 K5 K100
LD     T70
OR     X10006	; 前上下测料上下气缸SET传感器
ANB
SET    M1917
RST    M1929
LD     M1917
ANI    M101	; 暂停
SET    M1918
MPS
AND<>  D206 K0	; 前吸爪1料状态
RST    Y10201	; 前上下测料真空吸1电磁阀
SET    Y10202	; 前上下测料破真空1电磁阀
MRD
AND<>  D207 K0	; 前吸爪2料状态
RST    Y10205	; 前上下测料真空吸2电磁阀
SET    Y10206	; 前上下测料破真空2电磁阀
MPP
RST    M1917
LD     M1918
TMR    T27 K4 K100
AND    T27
SET    M1919
RST    Y10137	; 前上下测料上下电磁阀
RST    Y10202	; 前上下测料破真空1电磁阀
RST    Y10206	; 前上下测料破真空2电磁阀
RST    M1918

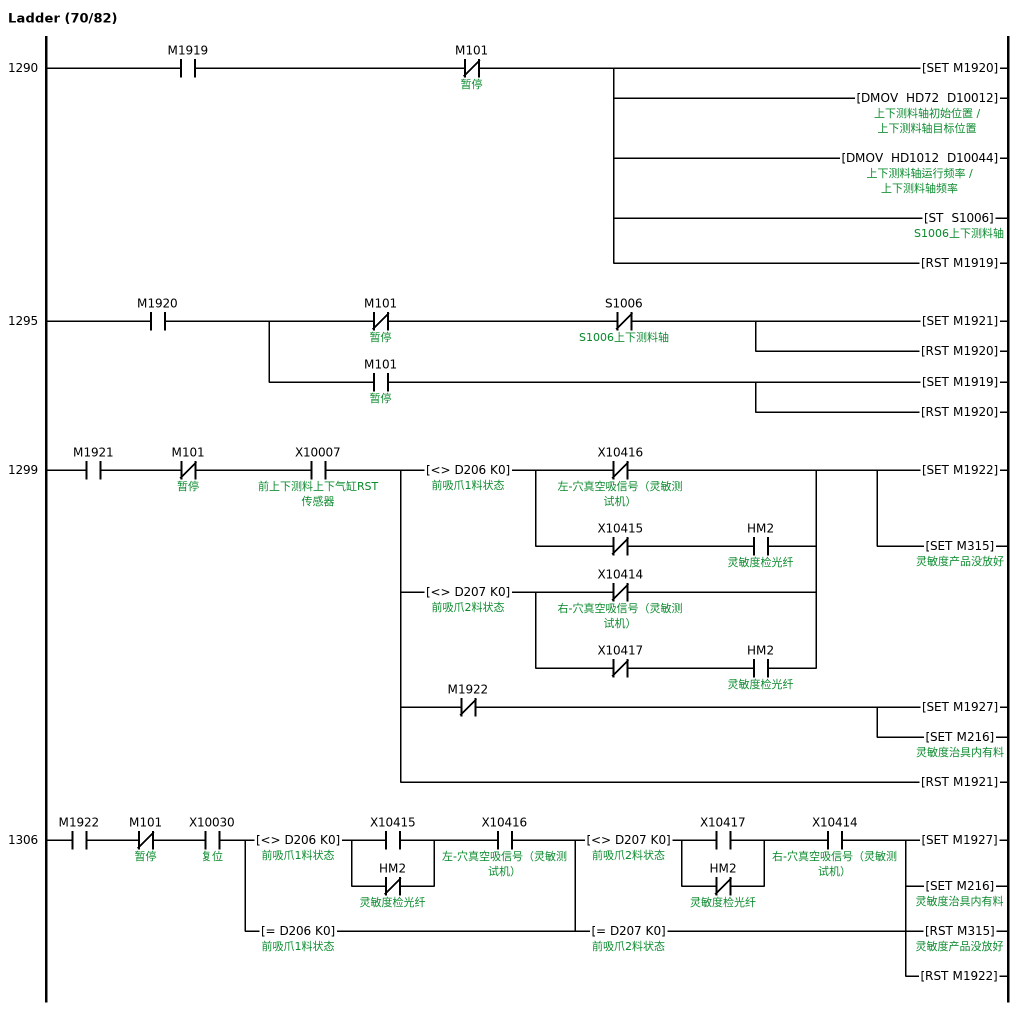
LD     M1919
ANI    M101	; 暂停
SET    M1920
DMOV   HD72 D10012	; 上下测料轴初始位置 / 上下测料轴目标位置
DMOV   HD1012 D10044	; 上下测料轴运行频率 / 上下测料轴频率
ST     S1006	; S1006上下测料轴
RST    M1919
LD     M1920
MPS
ANI    M101	; 暂停
ANI    S1006	; S1006上下测料轴
SET    M1921
RST    M1920
MPP
AND    M101	; 暂停
SET    M1919
RST    M1920
LD     M1921
ANI    M101	; 暂停
AND    X10007	; 前上下测料上下气缸RST传感器
MPS
LD<>   D206 K0	; 前吸爪1料状态
LDI    X10416	; 左-穴真空吸信号（灵敏测试机）
LDI    X10415
AND    HM2	; 灵敏度检光纤
ORB
ANB
LD<>   D207 K0	; 前吸爪2料状态
LDI    X10414	; 右-穴真空吸信号（灵敏测试机）
LDI    X10417
AND    HM2	; 灵敏度检光纤
ORB
ANB
ORB
ANB
SET    M1922
SET    M315	; 灵敏度产品没放好
MRD
ANI    M1922
SET    M1927
SET    M216	; 灵敏度治具内有料
MPP
RST    M1921
LD     M1922
ANI    M101	; 暂停
AND    X10030	; 复位
LD<>   D206 K0	; 前吸爪1料状态
LD     X10415
ORI    HM2	; 灵敏度检光纤
ANB
AND    X10416	; 左-穴真空吸信号（灵敏测试机）
OR=    D206 K0	; 前吸爪1料状态
ANB
LD<>   D207 K0	; 前吸爪2料状态
LD     X10417
ORI    HM2	; 灵敏度检光纤
ANB
AND    X10414	; 右-穴真空吸信号（灵敏测试机）
OR=    D207 K0	; 前吸爪2料状态
ANB
SET    M1927
SET    M216	; 灵敏度治具内有料
RST    M315	; 灵敏度产品没放好
RST    M1922

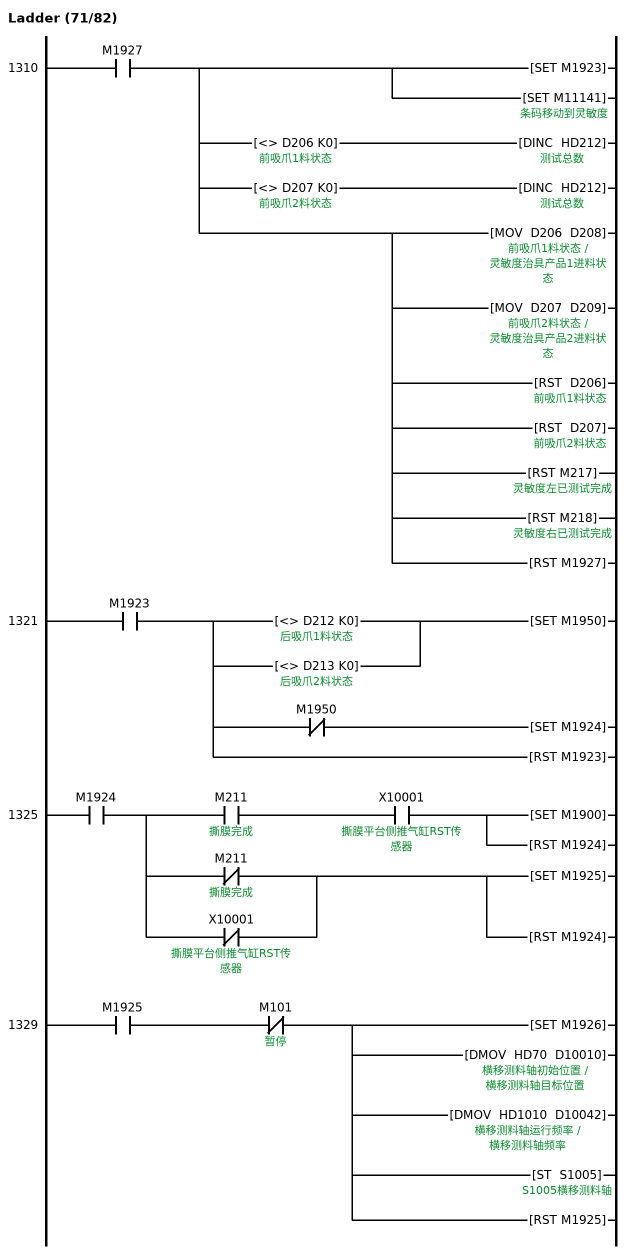
LD     M1927
SET    M1923
SET    M11141	; 条码移动到灵敏度
MPS
AND<>  D206 K0	; 前吸爪1料状态
DINC   HD212	; 测试总数
MRD
AND<>  D207 K0	; 前吸爪2料状态
DINC   HD212	; 测试总数
MPP
MOV    D206 D208	; 前吸爪1料状态 / 灵敏度治具产品1进料状态
MOV    D207 D209	; 前吸爪2料状态 / 灵敏度治具产品2进料状态
RST    D206	; 前吸爪1料状态
RST    D207	; 前吸爪2料状态
RST    M217	; 灵敏度左已测试完成
RST    M218	; 灵敏度右已测试完成
RST    M1927
LD     M1923
MPS
LD<>   D212 K0	; 后吸爪1料状态
OR<>   D213 K0	; 后吸爪2料状态
ANB
SET    M1950
MRD
ANI    M1950
SET    M1924
MPP
RST    M1923
LD     M1924
MPS
AND    M211	; 撕膜完成
AND    X10001	; 撕膜平台侧推气缸RST传感器
SET    M1900
RST    M1924
MPP
LDI    M211	; 撕膜完成
ORI    X10001	; 撕膜平台侧推气缸RST传感器
ANB
SET    M1925
RST    M1924
LD     M1925
ANI    M101	; 暂停
SET    M1926
DMOV   HD70 D10010	; 横移测料轴初始位置 / 横移测料轴目标位置
DMOV   HD1010 D10042	; 横移测料轴运行频率 / 横移测料轴频率
ST     S1005	; S1005横移测料轴
RST    M1925

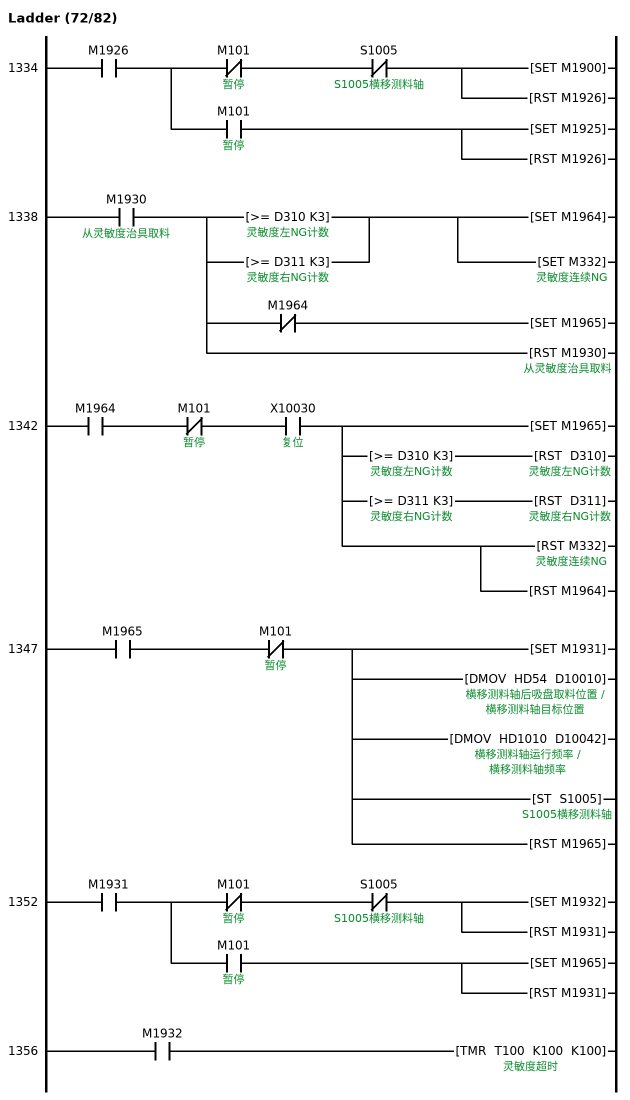
LD     M1926
MPS
ANI    M101	; 暂停
ANI    S1005	; S1005横移测料轴
SET    M1900
RST    M1926
MPP
AND    M101	; 暂停
SET    M1925
RST    M1926
LD     M1930	; 从灵敏度治具取料
MPS
LD>=   D310 K3	; 灵敏度左NG计数
OR>=   D311 K3	; 灵敏度右NG计数
ANB
SET    M1964
SET    M332	; 灵敏度连续NG
MRD
ANI    M1964
SET    M1965
MPP
RST    M1930	; 从灵敏度治具取料
LD     M1964
ANI    M101	; 暂停
AND    X10030	; 复位
SET    M1965
MPS
AND>=  D310 K3	; 灵敏度左NG计数
RST    D310	; 灵敏度左NG计数
MRD
AND>=  D311 K3	; 灵敏度右NG计数
RST    D311	; 灵敏度右NG计数
MPP
RST    M332	; 灵敏度连续NG
RST    M1964
LD     M1965
ANI    M101	; 暂停
SET    M1931
DMOV   HD54 D10010	; 横移测料轴后吸盘取料位置 / 横移测料轴目标位置
DMOV   HD1010 D10042	; 横移测料轴运行频率 / 横移测料轴频率
ST     S1005	; S1005横移测料轴
RST    M1965
LD     M1931
MPS
ANI    M101	; 暂停
ANI    S1005	; S1005横移测料轴
SET    M1932
RST    M1931
MPP
AND    M101	; 暂停
SET    M1965
RST    M1931
LD     M1932
TMR    T100 K100 K100	; 灵敏度超时

